{attribute 'qualified_only'}
VAR_GLOBAL
	bYellowButton 	AT %I*:BOOL;
	bBlueButton		AT %I* :BOOL;
	
	bGreenLight		AT %Q*:BOOL;
	bRedLight		AT %Q*:BOOL;
	
	iUltraschallSensor AT %I*:INT;
END_VAR

(* stored: Version 1.1.0.1, ProductVersion 3.1.4024.13
   GVL IO: Id {105c3da9-d06b-4696-96d7-893d47d8308e} *)
